{attribute 'qualified_only'}
{attribute 'strict'}
TYPE CmdServo :
(
	None,
	Enable,
	Disable,
	Reset,
	Home,
	StartMove,
	Stop,
	Jog
);
END_TYPE

(* stored: Version 1.1.0.1, ProductVersion 3.1.4022.11
   DUT CmdServo: Id {b50a4ebe-506e-42ed-8fd3-c0e420b2b190} *)
